TEXTLIST languageSupport
  axesAvailable = 'PLC Axes available: %d' | Test: 'Alt language'
  velocity = 'Velocity:'
  actposition = 'Actual Position:'
  enable = 'Enable Axis'
  enFW = 'Enable Forward'
  enBW = 'Enable Backward'
  axisSel = 'Axis Selected:'
  actVelocity = 'Actual Velocity:'
  errID = 'Error ID:'
  bEnabled = 'Axis Enabled'
  bWarning = 'Warning'
  bBusy = 'Busy'
  bDone = 'Command Done'
  bHomed = 'Calibrated'
  bFwEnabled = 'Fwd movement enabled'
  bBwEnabled = 'Bwd movement enabled'
  bError = 'Error'
  fVelocity = 'Target Velocity:' | Test: 'Geschwindigkeit:'
  fAcceleration = 'Target Accel.:'
  fDeceleration = 'Target Decel.:'
  fPosition = 'Target Position:'
  moveAbsolute = 'Absolute position move'
  toggle = 'Toggle'
  moveVelocity = 'Constant velocity move'
  bExecute = 'Motion function executed'
  moveRelative = 'Relative position move'
  moveModulo = 'Modulo position move'
  reset = 'Reset axis'
  stop = 'Stop motion'
  jogBw = 'Jog Backward'
  jogFw = 'Jog Forward'
  bGeared = 'In Gear'
  masterGear = 'Master Axis'
  gearRatio = 'Gear Ratio'
  gearIn = 'Gear In'
  gearOut = 'Gear Out'
  homeSensorNeg = 'Home to Sensor (Neg)'
  homeSensorPos = 'Home to Sensor (Pos)'
   = ''
END_TEXTLIST

(* stored: Version 1.1.0.1, ProductVersion 3.1.4024.2
   TextList languageSupport: Id {5d3fdc2f-5bea-44d3-8108-bdef8127e821} *)
